FUNCTION_BLOCK FB_Dispenser_1
VAR_INPUT
    bEnable      : BOOL;
    bExecute     : BOOL;
    nDispenceGram: REAL;
END_VAR

VAR_IN_OUT
    ax : AXIS_REF;  // Achsen Referenz
END_VAR

VAR_OUTPUT
    eStatus : State;
    bDone   : BOOL;
END_VAR

VAR
    fbPower        : MC_Power;
    fbMoveDistance : MC_MoveRelative;
    fbHalt         : MC_Halt;
    bAxPower       : BOOL;
    bAxMove        : BOOL;
    bHalt          : BOOL;
    nDistance      : REAL;
	nVelocity 	   : REAL := 50;
    eState_dispenser : INT := 0;
    doneTimer      : TON;
END_VAR

// Berechne die Bewegungsdistanz
nDistance := (nDispenceGram * 50);

// Achse updaten
ax.ReadStatus();

// Achsenfreigabe (Power) aufrufen
fbPower(Axis := ax, Enable := bAxPower, Enable_Positive := TRUE, Enable_Negative := TRUE);

// Bewegungsbefehl aufrufen
fbMoveDistance(Axis := ax, Execute := bAxMove, Distance := nDistance, Velocity := nVelocity);

// Haltbefehl aufrufen
fbHalt(Axis := ax, Execute := bHalt);

IF NOT bEnable THEN
    eState_dispenser := 0;
    eStatus := State.Off;
    bAxPower := FALSE;
    bAxMove := FALSE;
    bHalt := TRUE;
    bDone := FALSE;
ELSE
    CASE eState_dispenser OF
        0: // Off
            eStatus := State.Off;
            bAxPower := FALSE;
            bAxMove := FALSE;
            bHalt := TRUE;
            bDone := FALSE;
            IF bEnable THEN
                eState_dispenser := 1;
            END_IF

        1: // Powering up
            eStatus := State.Init;
            bAxPower := TRUE;
            IF fbPower.Status THEN
                eState_dispenser := 2;
            END_IF

        2: // Ready
            eStatus := State.Ready;
            bAxMove := FALSE;
            bHalt := FALSE;
            bDone := FALSE;
            IF bExecute THEN
                eState_dispenser := 3;
            END_IF

        3: // Production
            eStatus := State.Production;
            bAxMove := TRUE;
            bHalt := FALSE;
            
            IF fbMoveDistance.Done THEN
                bAxMove := FALSE;
                bDone := TRUE;
				eStatus := State.Done;
                eState_dispenser := 4;
            END_IF

        4: // Done, waiting to reset
			doneTimer(IN := TRUE, PT := T#2S);
            IF doneTimer.Q THEN
                doneTimer.IN := FALSE;
                bDone := FALSE;
                eState_dispenser := 2; // Zurück zu Ready
            END_IF
    END_CASE
END_IF

END_FUNCTION_BLOCK

(* stored: Version 1.1.0.1, ProductVersion 3.1.4024.12
   POU FB_Dispenser_1: Id {ec717c8d-62b6-4e1c-a2c4-d801fa8f7c18}, SpecialFunc None *)
